// TIA Portal V15.1 export
// export: Created 2024-06-21T08:41:01.6474151Z, ExportSetting WithDefaults, DisplayName Totally Integrated Automation Portal, DisplayVersion V15.1 Update 5, DisplayName TIA Portal Openness, DisplayVersion V15.1 Update 5, DisplayName SINAMICS Startdrive Advanced, DisplayVersion V15.1, DisplayName G130, G150, S120, S150, SINAMICS MV, S210, DisplayVersion V15.1, DisplayName G110M, G120, G120C, G120D, G120P, DisplayVersion V15.1, DisplayName STEP 7 Professional, DisplayVersion V15.1 Update 5, DisplayName STEP 7 Safety, DisplayVersion V15.1, DisplayName WinCC Professional, DisplayVersion V15.1 Update 5, DisplayName SIMATIC Visualization Architect, DisplayVersion V15.1
FUNCTION_BLOCK "LActiveShift"   // FB1800, FBD
TITLE = LActifShift
{ S7_Optimized_Access := 'FALSE' }
AUTHOR : VCC
FAMILY : Supervis
NAME : LActShif
VERSION : 1.0
// ================================================================================
// Module used to give which shift is active with the calendar variable of PLC
// Morning shift: start - stop is defined by HMI
// Evening shift: start - stop is defined by HMI
// Night shift  : start - stop is defined by HMI
// ================================================================================
// stored: AutoNumber false, IsIECCheckEnabled false, SetENOAutomatically False, UDAEnableTagReadback false
   VAR_OUTPUT
      O_MorningShift { ExternalAccessible := 'False'; ExternalVisible := 'False'; ExternalWritable := 'False'} : Bool;   // Morning shift
      O_EveningShift { ExternalAccessible := 'False'; ExternalVisible := 'False'; ExternalWritable := 'False'} : Bool;   // Evening shift
      O_NightShift { ExternalAccessible := 'False'; ExternalVisible := 'False'; ExternalWritable := 'False'} : Bool;   // NightShift
      O_NewShift { ExternalAccessible := 'False'; ExternalVisible := 'False'; ExternalWritable := 'False'} : Bool;   // NewShift / Morning shift
      O_ShiftOverview { ExternalAccessible := 'False'; ExternalVisible := 'False'; ExternalWritable := 'False'} : Struct   // Overview Active Shift
         MorningShift_Day1 { ExternalAccessible := 'False'; ExternalVisible := 'False'; ExternalWritable := 'False'} : Bool;   // Morning Shift of Day 1 (Monday)
         EveningShift_Day1 { ExternalAccessible := 'False'; ExternalVisible := 'False'; ExternalWritable := 'False'} : Bool;   // Evening Shift of Day 1 (Monday)
         NightShift_Day1 { ExternalAccessible := 'False'; ExternalVisible := 'False'; ExternalWritable := 'False'} : Bool;   // Night Shift of Day 1 (Monday-Tuesday)
         MorningShift_Day2 { ExternalAccessible := 'False'; ExternalVisible := 'False'; ExternalWritable := 'False'} : Bool;   // Morning Shift of Day 2 (Tuesday)
         EveningShift_Day2 { ExternalAccessible := 'False'; ExternalVisible := 'False'; ExternalWritable := 'False'} : Bool;   // Evening Shift of Day 2 (Tuesday)
         NightShift_Day2 { ExternalAccessible := 'False'; ExternalVisible := 'False'; ExternalWritable := 'False'} : Bool;   // Night Shift of Day 2 (Tuesday-Wednesday)
         MorningShift_Day3 { ExternalAccessible := 'False'; ExternalVisible := 'False'; ExternalWritable := 'False'} : Bool;   // Morning Shift of Day 3 (Wednesday)
         EveningShift_Day3 { ExternalAccessible := 'False'; ExternalVisible := 'False'; ExternalWritable := 'False'} : Bool;   // Evening Shift of Day 3 (Wednesday)
         NightShift_Day3 { ExternalAccessible := 'False'; ExternalVisible := 'False'; ExternalWritable := 'False'} : Bool;   // night Shift of Day 3 (Wednesday-Thursday)
         MorningShift_Day4 { ExternalAccessible := 'False'; ExternalVisible := 'False'; ExternalWritable := 'False'} : Bool;   // Morning Shift of Day 4 (Thursday)
         EveningShift_Day4 { ExternalAccessible := 'False'; ExternalVisible := 'False'; ExternalWritable := 'False'} : Bool;   // Evening Shift of Day 4 (Thursday)
         NightShift_Day4 { ExternalAccessible := 'False'; ExternalVisible := 'False'; ExternalWritable := 'False'} : Bool;   // Night Shift of Day 4 (Thursday-Friday)
         MorningShift_Day5 { ExternalAccessible := 'False'; ExternalVisible := 'False'; ExternalWritable := 'False'} : Bool;   // Morning Shift of Day 5 (Friday)
         EveningShift_Day5 { ExternalAccessible := 'False'; ExternalVisible := 'False'; ExternalWritable := 'False'} : Bool;   // Evening Shift of Day 5 (Friday)
         NightShift_Day5 { ExternalAccessible := 'False'; ExternalVisible := 'False'; ExternalWritable := 'False'} : Bool;   // Night Shift of Day 5 (Friday-Saturday)
         MorningShift_Day6 { ExternalAccessible := 'False'; ExternalVisible := 'False'; ExternalWritable := 'False'} : Bool;   // Morning Shift of Day 6 (Saturday)
         EveningShift_Day6 { ExternalAccessible := 'False'; ExternalVisible := 'False'; ExternalWritable := 'False'} : Bool;   // Evening Shift of Day 6 (Saturday)
         NightShift_Day6 { ExternalAccessible := 'False'; ExternalVisible := 'False'; ExternalWritable := 'False'} : Bool;   // Night Shift of Day 6 (Saturday-Sunday)
         MorningShift_Day7 { ExternalAccessible := 'False'; ExternalVisible := 'False'; ExternalWritable := 'False'} : Bool;   // Morning Shift of Day 7 (Sunday)
         EveningShift_Day7 { ExternalAccessible := 'False'; ExternalVisible := 'False'; ExternalWritable := 'False'} : Bool;   // Evening Shift of Day 7 (Sunday)
         NightShift_Day7 { ExternalAccessible := 'False'; ExternalVisible := 'False'; ExternalWritable := 'False'} : Bool;   // night Shift of Day 7 (Sunday-Monday)
      END_STRUCT;
      H_IAnim { ExternalAccessible := 'False'; ExternalVisible := 'False'; ExternalWritable := 'False'} : Word;   // HMI Animation of the icon
   END_VAR
   VAR DB_SPECIFIC
      H_In : Struct   // HMI
         StartMorningDay1 : Real := 5.15;   // Start time of morning shift - Day 1
         StartEveningDay1 : Real := 13.15;   // Start time of evening shift - Day 1
         StartNightDay1 : Real := 21.15;   // Start time of night shift - Day 1
         StartMorningDay2 : Real := 5.15;   // Start time of morning shift - Day 2
         StartEveningDay2 : Real := 13.15;   // Start time of evening shift - Day 2
         StartNightDay2 : Real := 21.15;   // Start time of night shift - Day 2
         StartMorningDay3 : Real := 5.15;   // Start time of morning shift - Day 3
         StartEveningDay3 : Real := 13.15;   // Start time of evening shift - Day 3
         StartNightDay3 : Real := 21.15;   // Start time of night shift - Day 3
         StartMorningDay4 : Real := 5.15;   // Start time of morning shift - Day 4
         StartEveningDay4 : Real := 13.15;   // Start time of evening shift - Day 4
         StartNightDay4 : Real := 21.15;   // Start time of night shift - Day 4
         StartMorningDay5 : Real := 5.15;   // Start time of morning shift - Day 5
         StartEveningDay5 : Real := 12.25;   // Start time of evening shift - Day 5
         StartNightDay5 : Real := 19.35;   // Start time of night shift - Day 5
         StartMorningDay6 : Real := 5.15;   // Start time of morning shift - Day 6
         StartEveningDay6 : Real := 13.15;   // Start time of evening shift - Day 6
         StartNightDay6 : Real := 21.15;   // Start time of night shift - Day 6
         StartMorningDay7 : Real := 5.15;   // Start time of morning shift - Day 7
         StartEveningDay7 : Real := 13.15;   // Start time of evening shift - Day 7
         StartNightDay7 : Real := 21.15;   // Start time of night shift - Day 7
      END_STRUCT;
      H_Out : Struct   // HMI
         Anim : Word;   // HMI Animation of the object
         DBnr : Int;   // HMI Animation DB number
      END_STRUCT;
      MorningShift_Day1 { ExternalAccessible := 'False'; ExternalVisible := 'False'; ExternalWritable := 'False'} : Bool;   // Morning Shift of Day 1 (Monday)
      EveningShift_Day1 { ExternalAccessible := 'False'; ExternalVisible := 'False'; ExternalWritable := 'False'} : Bool;   // Evening Shift of Day 1 (Monday)
      NightShift_Day1 { ExternalAccessible := 'False'; ExternalVisible := 'False'; ExternalWritable := 'False'} : Bool;   // Night Shift of Day 1 (Monday-Tuesday)
      MorningShift_Day2 { ExternalAccessible := 'False'; ExternalVisible := 'False'; ExternalWritable := 'False'} : Bool;   // Morning Shift of Day 2 (Tuesday)
      EveningShift_Day2 { ExternalAccessible := 'False'; ExternalVisible := 'False'; ExternalWritable := 'False'} : Bool;   // Evening Shift of Day 2 (Tuesday)
      NightShift_Day2 { ExternalAccessible := 'False'; ExternalVisible := 'False'; ExternalWritable := 'False'} : Bool;   // Night Shift of Day 2 (Tuesday-Wednesday)
      MorningShift_Day3 { ExternalAccessible := 'False'; ExternalVisible := 'False'; ExternalWritable := 'False'} : Bool;   // Morning Shift of Day 3 (Wednesday)
      EveningShift_Day3 { ExternalAccessible := 'False'; ExternalVisible := 'False'; ExternalWritable := 'False'} : Bool;   // Evening Shift of Day 3 (Wednesday)
      NightShift_Day3 { ExternalAccessible := 'False'; ExternalVisible := 'False'; ExternalWritable := 'False'} : Bool;   // night Shift of Day 3 (Wednesday-Thursday)
      MorningShift_Day4 { ExternalAccessible := 'False'; ExternalVisible := 'False'; ExternalWritable := 'False'} : Bool;   // Morning Shift of Day 4 (Thursday)
      EveningShift_Day4 { ExternalAccessible := 'False'; ExternalVisible := 'False'; ExternalWritable := 'False'} : Bool;   // Evening Shift of Day 4 (Thursday)
      NightShift_Day4 { ExternalAccessible := 'False'; ExternalVisible := 'False'; ExternalWritable := 'False'} : Bool;   // Night Shift of Day 4 (Thursday-Friday)
      MorningShift_Day5 { ExternalAccessible := 'False'; ExternalVisible := 'False'; ExternalWritable := 'False'} : Bool;   // Morning Shift of Day 5 (Friday)
      EveningShift_Day5 { ExternalAccessible := 'False'; ExternalVisible := 'False'; ExternalWritable := 'False'} : Bool;   // Evening Shift of Day 5 (Friday)
      NightShift_Day5 { ExternalAccessible := 'False'; ExternalVisible := 'False'; ExternalWritable := 'False'} : Bool;   // Night Shift of Day 5 (Friday-Saturday)
      MorningShift_Day6 { ExternalAccessible := 'False'; ExternalVisible := 'False'; ExternalWritable := 'False'} : Bool;   // Morning Shift of Day 6 (Saturday)
      EveningShift_Day6 { ExternalAccessible := 'False'; ExternalVisible := 'False'; ExternalWritable := 'False'} : Bool;   // Evening Shift of Day 6 (Saturday)
      NightShift_Day6 { ExternalAccessible := 'False'; ExternalVisible := 'False'; ExternalWritable := 'False'} : Bool;   // Night Shift of Day 6 (Saturday-Sunday)
      MorningShift_Day7 { ExternalAccessible := 'False'; ExternalVisible := 'False'; ExternalWritable := 'False'} : Bool;   // Morning Shift of Day 7 (Sunday)
      EveningShift_Day7 { ExternalAccessible := 'False'; ExternalVisible := 'False'; ExternalWritable := 'False'} : Bool;   // Evening Shift of Day 7 (Sunday)
      NightShift_Day7 { ExternalAccessible := 'False'; ExternalVisible := 'False'; ExternalWritable := 'False'} : Bool;   // night Shift of Day 7 (Sunday-Monday)
      MorningShift { ExternalAccessible := 'False'; ExternalVisible := 'False'; ExternalWritable := 'False'} : Bool;   // Morning shift
      EveningShift { ExternalAccessible := 'False'; ExternalVisible := 'False'; ExternalWritable := 'False'} : Bool;   // Evening shift
      NightShift { ExternalAccessible := 'False'; ExternalVisible := 'False'; ExternalWritable := 'False'} : Bool;   // NightShift
      NewShift { ExternalAccessible := 'False'; ExternalVisible := 'False'; ExternalWritable := 'False'} : Bool;   // NewShift / Morning shift
      NewMorningShiftTrig { ExternalAccessible := 'False'; ExternalVisible := 'False'; ExternalWritable := 'False'} : Bool;   // Trigger for New Morning shift / Morning shift
      NewEveningShiftTrig { ExternalAccessible := 'False'; ExternalVisible := 'False'; ExternalWritable := 'False'} : Bool;   // Trigger for New Evening shift / Evening shift
      NewNightShiftTrig { ExternalAccessible := 'False'; ExternalVisible := 'False'; ExternalWritable := 'False'} : Bool;   // Trigger for New NightShift / NightShift
      Day1 { ExternalAccessible := 'False'; ExternalVisible := 'False'; ExternalWritable := 'False'} : Bool;   // Day 1 = Monday
      Day2 { ExternalAccessible := 'False'; ExternalVisible := 'False'; ExternalWritable := 'False'} : Bool;   // Day 2 = Tuesday
      Day3 { ExternalAccessible := 'False'; ExternalVisible := 'False'; ExternalWritable := 'False'} : Bool;   // Day 3 = Wednesday
      Day4 { ExternalAccessible := 'False'; ExternalVisible := 'False'; ExternalWritable := 'False'} : Bool;   // Day 4 = Thursday
      Day5 { ExternalAccessible := 'False'; ExternalVisible := 'False'; ExternalWritable := 'False'} : Bool;   // Day 5 = Friday
      Day6 { ExternalAccessible := 'False'; ExternalVisible := 'False'; ExternalWritable := 'False'} : Bool;   // Day 6 = Saturday
      Day7 { ExternalAccessible := 'False'; ExternalVisible := 'False'; ExternalWritable := 'False'} : Bool;   // Day 7 = Sunday
      Day1_Int_Morning { ExternalAccessible := 'False'; ExternalVisible := 'False'; ExternalWritable := 'False'} : Int := 515;   // Start integer of morning shift - Day 1
      Day1_Int_Evening { ExternalAccessible := 'False'; ExternalVisible := 'False'; ExternalWritable := 'False'} : Int := 1315;   // Start integer of evening shift - Day 1
      Day1_Int_Night { ExternalAccessible := 'False'; ExternalVisible := 'False'; ExternalWritable := 'False'} : Int := 2115;   // Start integer of night shift - Day 1
      Day2_Int_Morning { ExternalAccessible := 'False'; ExternalVisible := 'False'; ExternalWritable := 'False'} : Int := 515;   // Start integer of morning shift - Day 2
      Day2_Int_Evening { ExternalAccessible := 'False'; ExternalVisible := 'False'; ExternalWritable := 'False'} : Int := 1315;   // Start integer of evening shift - Day 2
      Day2_Int_Night { ExternalAccessible := 'False'; ExternalVisible := 'False'; ExternalWritable := 'False'} : Int := 2115;   // Start integer of night shift - Day 2
      Day3_Int_Morning { ExternalAccessible := 'False'; ExternalVisible := 'False'; ExternalWritable := 'False'} : Int := 515;   // Start integer of morning shift - Day 3
      Day3_Int_Evening { ExternalAccessible := 'False'; ExternalVisible := 'False'; ExternalWritable := 'False'} : Int := 1315;   // Start integer of evening shift - Day 3
      Day3_Int_Night { ExternalAccessible := 'False'; ExternalVisible := 'False'; ExternalWritable := 'False'} : Int := 2115;   // Start integer of night shift - Day 3
      Day4_Int_Morning { ExternalAccessible := 'False'; ExternalVisible := 'False'; ExternalWritable := 'False'} : Int := 515;   // Start integer of morning shift - Day 4
      Day4_Int_Evening { ExternalAccessible := 'False'; ExternalVisible := 'False'; ExternalWritable := 'False'} : Int := 1315;   // Start integer of evening shift - Day 4
      Day4_Int_Night { ExternalAccessible := 'False'; ExternalVisible := 'False'; ExternalWritable := 'False'} : Int := 2115;   // Start integer of night shift - Day 4
      Day5_Int_Morning { ExternalAccessible := 'False'; ExternalVisible := 'False'; ExternalWritable := 'False'} : Int := 515;   // Start integer of morning shift - Day 5
      Day5_Int_Evening { ExternalAccessible := 'False'; ExternalVisible := 'False'; ExternalWritable := 'False'} : Int := 1225;   // Start integer of evening shift - Day 5
      Day5_Int_Night { ExternalAccessible := 'False'; ExternalVisible := 'False'; ExternalWritable := 'False'} : Int := 1935;   // Start integer of night shift - Day 5
      Day6_Int_Morning { ExternalAccessible := 'False'; ExternalVisible := 'False'; ExternalWritable := 'False'} : Int := 515;   // Start integer of morning shift - Day 6
      Day6_Int_Evening { ExternalAccessible := 'False'; ExternalVisible := 'False'; ExternalWritable := 'False'} : Int := 1315;   // Start integer of evening shift - Day 6
      Day6_Int_Night { ExternalAccessible := 'False'; ExternalVisible := 'False'; ExternalWritable := 'False'} : Int := 2115;   // Start integer of night shift - Day 6
      Day7_Int_Morning { ExternalAccessible := 'False'; ExternalVisible := 'False'; ExternalWritable := 'False'} : Int := 515;   // Start integer of morning shift - Day 7
      Day7_Int_Evening { ExternalAccessible := 'False'; ExternalVisible := 'False'; ExternalWritable := 'False'} : Int := 1315;   // Start integer of evening shift - Day 7
      Day7_Int_Night { ExternalAccessible := 'False'; ExternalVisible := 'False'; ExternalWritable := 'False'} : Int := 2115;   // Start integer of night shift - Day 7
      DBnr { ExternalAccessible := 'False'; ExternalVisible := 'False'; ExternalWritable := 'False'} : Int;   // HMI DB number
   END_VAR
   VAR_TEMP
      Temp1 : Real;
      Temp2 : Int;
   END_VAR
   VAR_TEMP   // added for the SCL form of the ladder/FBD networks
      _w1 : Bool;
      _w2 : Bool;
      _w3 : Bool;
   END_VAR
BEGIN

NETWORK
TITLE = **** 1 - Inputs **** DB number
// DB number
      L     DINO;
      T     #DBnr;

NETWORK
TITLE = **** 4.4 - Machine status - Calculated **** Copy time from HMI to integer
// Copy time from HMI to integer
//********************** Time day 1 *****************************
      L     #H_In.StartMorningDay1;  // Load Start time of morning shift - Day 1
      L     100.0;  // * 100
      *R;  // *
      RND;  // Conversion real to integer
      T     #Day1_Int_Morning;  // Load start time of morning shift = Day 1

      L     #H_In.StartEveningDay1;  // Load Start time of evening shift - Day 1
      L     100.0;  // * 100
      *R;  // *
      RND;  // Conversion real to integer
      T     #Day1_Int_Evening;  // Load start time of evening shift = Day 1

      L     #H_In.StartNightDay1;  // Load Start time of night shift - Day 1
      L     100.0;  // * 100
      *R;  // *
      RND;  // Conversion real to integer
      T     #Day1_Int_Night;  // Load start time of night shift = Day 1


//********************** Time day 2 *****************************
      L     #H_In.StartMorningDay2;  // Load Start time of morning shift - Day 2
      L     100.0;  // * 100
      *R;  // *
      RND;  // Conversion real to integer
      T     #Day2_Int_Morning;  // Load start time of morning shift = Day 2

      L     #H_In.StartEveningDay2;  // Load Start time of evening shift - Day 2
      L     100.0;  // * 100
      *R;  // *
      RND;  // Conversion real to integer
      T     #Day2_Int_Evening;  // Load start time of evening shift = Day 2

      L     #H_In.StartNightDay2;  // Load Start time of night shift - Day 2
      L     100.0;  // * 100
      *R;  // *
      RND;  // Conversion real to integer
      T     #Day2_Int_Night;  // Load start time of night shift = Day 2

//********************** Time day 3 *****************************
      L     #H_In.StartMorningDay3;  // Load Start time of morning shift - Day 3
      L     100.0;  // * 100
      *R;  // *
      RND;  // Conversion real to integer
      T     #Day3_Int_Morning;  // Load start time of morning shift = Day 3

      L     #H_In.StartEveningDay3;  // Load Start time of evening shift - Day 3
      L     100.0;  // * 100
      *R;  // *
      RND;  // Conversion real to integer
      T     #Day3_Int_Evening;  // Load start time of evening shift = Day 3

      L     #H_In.StartNightDay3;  // Load Start time of night shift - Day 3
      L     100.0;  // * 100
      *R;  // *
      RND;  // Conversion real to integer
      T     #Day3_Int_Night;  // Load start time of night shift = Day 3

//********************** Time day 4 *****************************
      L     #H_In.StartMorningDay4;  // Load Start time of morning shift - Day 4
      L     100.0;  // * 100
      *R;  // *
      RND;  // Conversion real to integer
      T     #Day4_Int_Morning;  // Load start time of morning shift = Day 4

      L     #H_In.StartEveningDay4;  // Load Start time of evening shift - Day 4
      L     100.0;  // * 100
      *R;  // *
      RND;  // Conversion real to integer
      T     #Day4_Int_Evening;  // Load start time of evening shift = Day 4

      L     #H_In.StartNightDay4;  // Load Start time of night shift - Day 4
      L     100.0;  // * 100
      *R;  // *
      RND;  // Conversion real to integer
      T     #Day4_Int_Night;  // Load start time of night shift = Day 4

//********************** Time day 5 *****************************
      L     #H_In.StartMorningDay5;  // Load Start time of morning shift - Day 5
      L     100.0;  // * 100
      *R;  // *
      RND;  // Conversion real to integer
      T     #Day5_Int_Morning;  // Load start time of morning shift = Day 5

      L     #H_In.StartEveningDay5;  // Load Start time of evening shift - Day 5
      L     100.0;  // * 100
      *R;  // *
      RND;  // Conversion real to integer
      T     #Day5_Int_Evening;  // Load start time of evening shift = Day 5

      L     #H_In.StartNightDay5;  // Load Start time of night shift - Day 5
      L     100.0;  // * 100
      *R;  // *
      RND;  // Conversion real to integer
      T     #Day5_Int_Night;  // Load start time of night shift = Day 5

//********************** Time day 6 *****************************
      L     #H_In.StartMorningDay6;  // Load Start time of morning shift - Day 6
      L     100.0;  // * 100
      *R;  // *
      RND;  // Conversion real to integer
      T     #Day6_Int_Morning;  // Load start time of morning shift = Day 6

      L     #H_In.StartEveningDay6;  // Load Start time of evening shift - Day 6
      L     100.0;  // * 100
      *R;  // *
      RND;  // Conversion real to integer
      T     #Day6_Int_Evening;  // Load start time of evening shift = Day 6

      L     #H_In.StartNightDay6;  // Load Start time of night shift - Day 6
      L     100.0;  // * 100
      *R;  // *
      RND;  // Conversion real to integer
      T     #Day6_Int_Night;  // Load start time of night shift = Day 6

//********************** Time day 7 *****************************
      L     #H_In.StartMorningDay7;  // Load Start time of morning shift - Day 7
      L     100.0;  // * 100
      *R;  // *
      RND;  // Conversion real to integer
      T     #Day7_Int_Morning;  // Load start time of morning shift = Day 7

      L     #H_In.StartEveningDay7;  // Load Start time of evening shift - Day 7
      L     100.0;  // * 100
      *R;  // *
      RND;  // Conversion real to integer
      T     #Day7_Int_Evening;  // Load start time of evening shift = Day 7

      L     #H_In.StartNightDay7;  // Load Start time of night shift - Day 7
      L     100.0;  // * 100
      *R;  // *
      RND;  // Conversion real to integer
      T     #Day7_Int_Night;  // Load start time of night shift = Day 7

REGION Network 3: **** 4.4 - Machine status - Calculated **** Morning Shift of Day 1
   // Morning Shift of Day 1
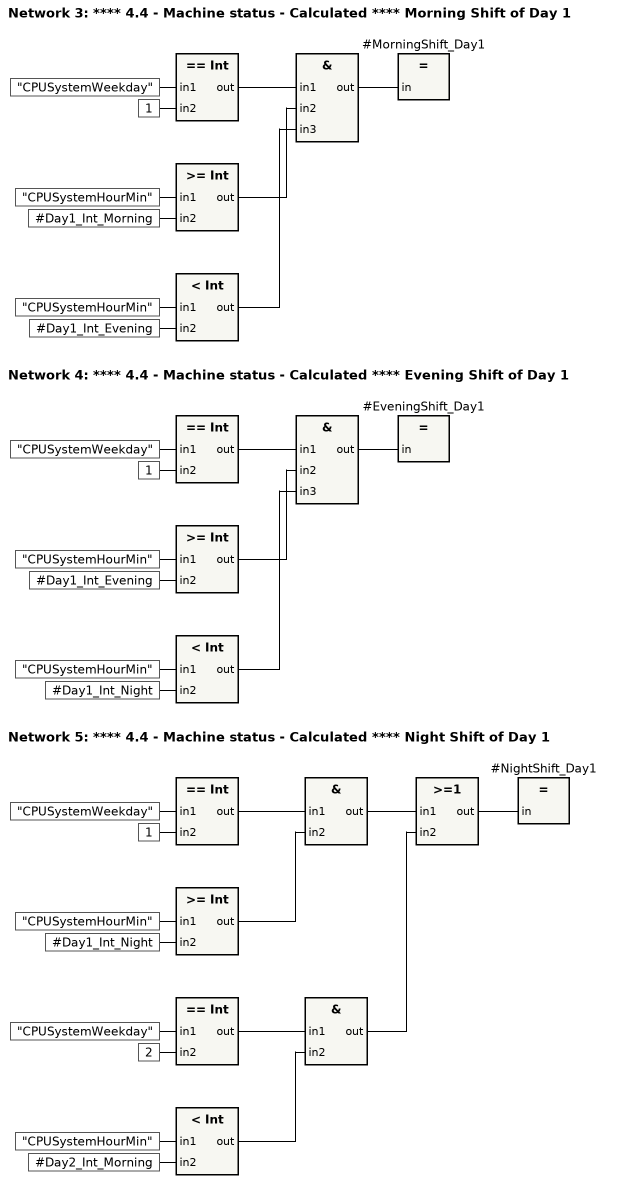
   #MorningShift_Day1 := ("CPUSystemWeekday" = 1) AND ("CPUSystemHourMin" >= #Day1_Int_Morning) AND ("CPUSystemHourMin" < #Day1_Int_Evening);
END_REGION

REGION Network 4: **** 4.4 - Machine status - Calculated **** Evening Shift of Day 1
   // Evening Shift of Day 1
   #EveningShift_Day1 := ("CPUSystemWeekday" = 1) AND ("CPUSystemHourMin" >= #Day1_Int_Evening) AND ("CPUSystemHourMin" < #Day1_Int_Night);
END_REGION

REGION Network 5: **** 4.4 - Machine status - Calculated **** Night Shift of Day 1
   // Night Shift of Day 1
   #NightShift_Day1 := (("CPUSystemWeekday" = 1) AND ("CPUSystemHourMin" >= #Day1_Int_Night)) OR (("CPUSystemWeekday" = 2) AND ("CPUSystemHourMin" < #Day2_Int_Morning));
END_REGION

REGION Network 6: **** 4.4 - Machine status - Calculated **** Morning Shift of Day 2
   // Morning Shift of Day 2
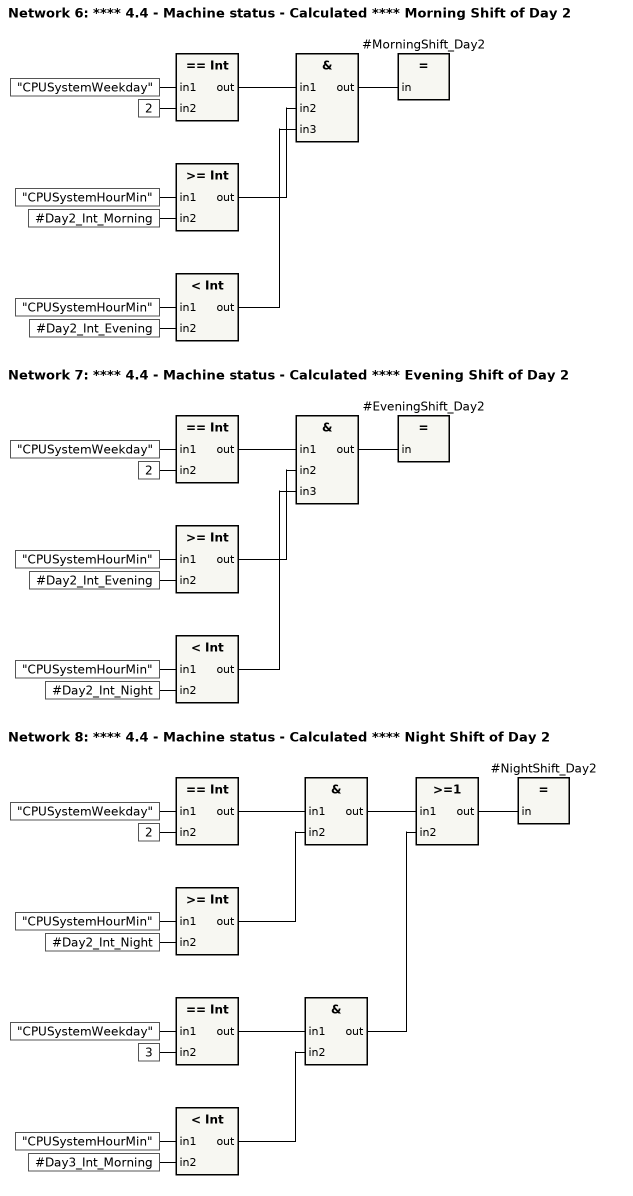
   #MorningShift_Day2 := ("CPUSystemWeekday" = 2) AND ("CPUSystemHourMin" >= #Day2_Int_Morning) AND ("CPUSystemHourMin" < #Day2_Int_Evening);
END_REGION

REGION Network 7: **** 4.4 - Machine status - Calculated **** Evening Shift of Day 2
   // Evening Shift of Day 2
   #EveningShift_Day2 := ("CPUSystemWeekday" = 2) AND ("CPUSystemHourMin" >= #Day2_Int_Evening) AND ("CPUSystemHourMin" < #Day2_Int_Night);
END_REGION

REGION Network 8: **** 4.4 - Machine status - Calculated **** Night Shift of Day 2
   // Night Shift of Day 2
   #NightShift_Day2 := (("CPUSystemWeekday" = 2) AND ("CPUSystemHourMin" >= #Day2_Int_Night)) OR (("CPUSystemWeekday" = 3) AND ("CPUSystemHourMin" < #Day3_Int_Morning));
END_REGION

REGION Network 9: **** 4.4 - Machine status - Calculated **** Morning Shift of Day 3
   // Morning Shift of Day 3
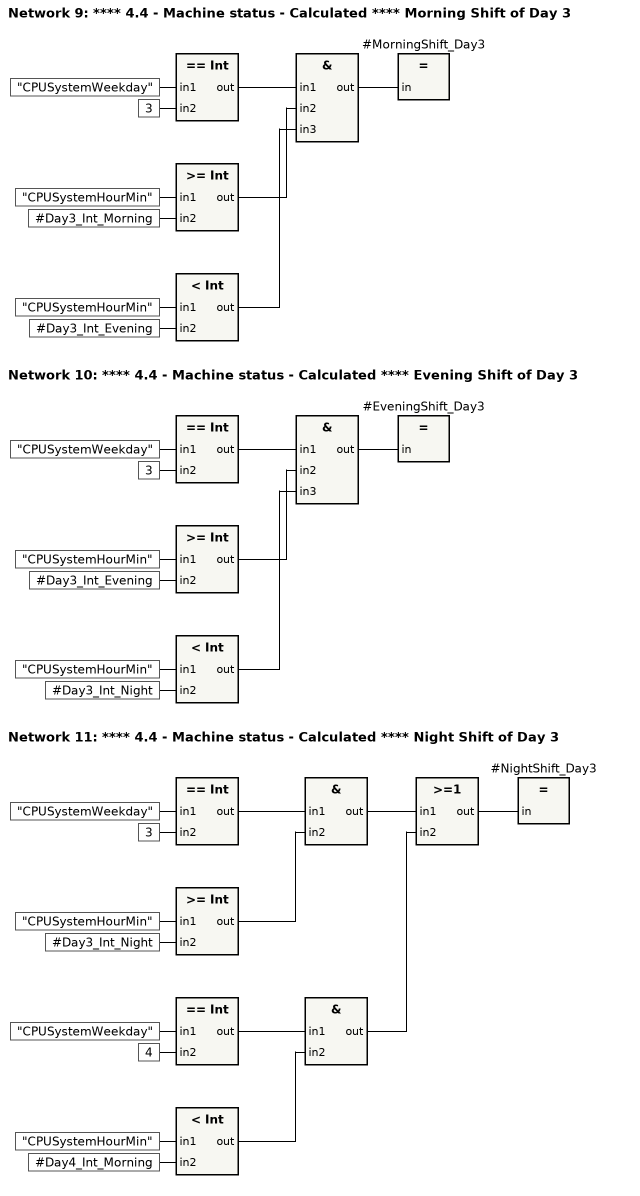
   #MorningShift_Day3 := ("CPUSystemWeekday" = 3) AND ("CPUSystemHourMin" >= #Day3_Int_Morning) AND ("CPUSystemHourMin" < #Day3_Int_Evening);
END_REGION

REGION Network 10: **** 4.4 - Machine status - Calculated **** Evening Shift of Day 3
   // Evening Shift of Day 3
   #EveningShift_Day3 := ("CPUSystemWeekday" = 3) AND ("CPUSystemHourMin" >= #Day3_Int_Evening) AND ("CPUSystemHourMin" < #Day3_Int_Night);
END_REGION

REGION Network 11: **** 4.4 - Machine status - Calculated **** Night Shift of Day 3
   // Night Shift of Day 3
   #NightShift_Day3 := (("CPUSystemWeekday" = 3) AND ("CPUSystemHourMin" >= #Day3_Int_Night)) OR (("CPUSystemWeekday" = 4) AND ("CPUSystemHourMin" < #Day4_Int_Morning));
END_REGION

REGION Network 12: **** 4.4 - Machine status - Calculated **** Morning Shift of Day 4
   // Morning Shift of Day 4
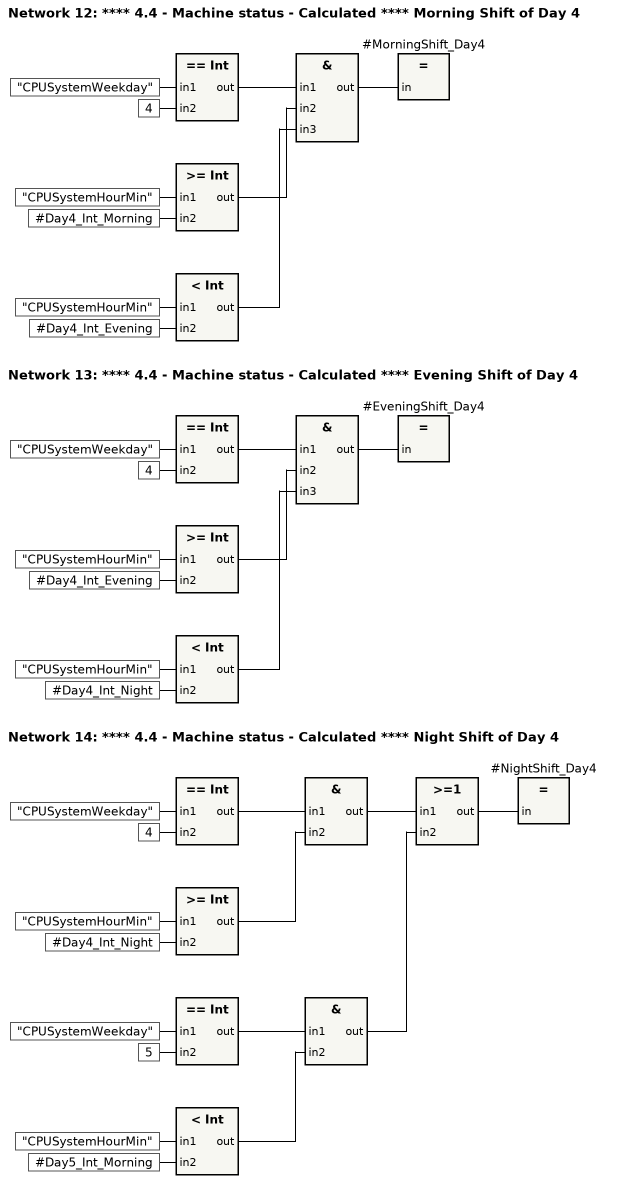
   #MorningShift_Day4 := ("CPUSystemWeekday" = 4) AND ("CPUSystemHourMin" >= #Day4_Int_Morning) AND ("CPUSystemHourMin" < #Day4_Int_Evening);
END_REGION

REGION Network 13: **** 4.4 - Machine status - Calculated **** Evening Shift of Day 4
   // Evening Shift of Day 4
   #EveningShift_Day4 := ("CPUSystemWeekday" = 4) AND ("CPUSystemHourMin" >= #Day4_Int_Evening) AND ("CPUSystemHourMin" < #Day4_Int_Night);
END_REGION

REGION Network 14: **** 4.4 - Machine status - Calculated **** Night Shift of Day 4
   // Night Shift of Day 4
   #NightShift_Day4 := (("CPUSystemWeekday" = 4) AND ("CPUSystemHourMin" >= #Day4_Int_Night)) OR (("CPUSystemWeekday" = 5) AND ("CPUSystemHourMin" < #Day5_Int_Morning));
END_REGION

REGION Network 15: **** 4.4 - Machine status - Calculated **** Morning Shift of Day 5
   // Morning Shift of Day 5
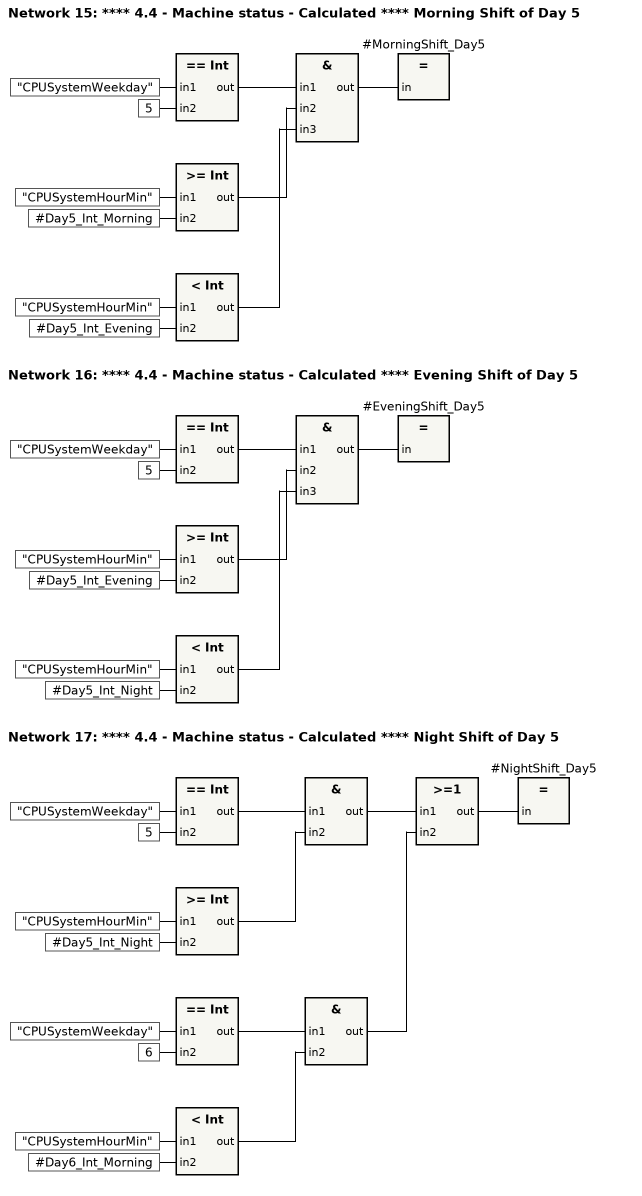
   #MorningShift_Day5 := ("CPUSystemWeekday" = 5) AND ("CPUSystemHourMin" >= #Day5_Int_Morning) AND ("CPUSystemHourMin" < #Day5_Int_Evening);
END_REGION

REGION Network 16: **** 4.4 - Machine status - Calculated **** Evening Shift of Day 5
   // Evening Shift of Day 5
   #EveningShift_Day5 := ("CPUSystemWeekday" = 5) AND ("CPUSystemHourMin" >= #Day5_Int_Evening) AND ("CPUSystemHourMin" < #Day5_Int_Night);
END_REGION

REGION Network 17: **** 4.4 - Machine status - Calculated **** Night Shift of Day 5
   // Night Shift of Day 5
   #NightShift_Day5 := (("CPUSystemWeekday" = 5) AND ("CPUSystemHourMin" >= #Day5_Int_Night)) OR (("CPUSystemWeekday" = 6) AND ("CPUSystemHourMin" < #Day6_Int_Morning));
END_REGION

REGION Network 18: **** 4.4 - Machine status - Calculated **** Morning Shift of Day 6
   // Morning Shift of Day 6
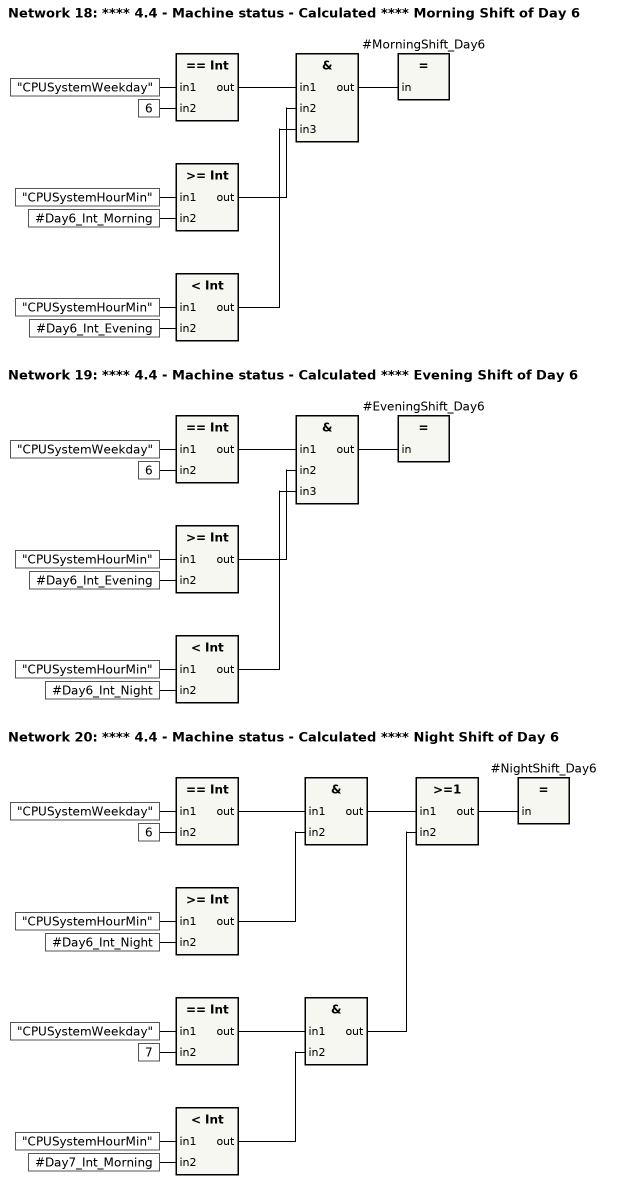
   #MorningShift_Day6 := ("CPUSystemWeekday" = 6) AND ("CPUSystemHourMin" >= #Day6_Int_Morning) AND ("CPUSystemHourMin" < #Day6_Int_Evening);
END_REGION

REGION Network 19: **** 4.4 - Machine status - Calculated **** Evening Shift of Day 6
   // Evening Shift of Day 6
   #EveningShift_Day6 := ("CPUSystemWeekday" = 6) AND ("CPUSystemHourMin" >= #Day6_Int_Evening) AND ("CPUSystemHourMin" < #Day6_Int_Night);
END_REGION

REGION Network 20: **** 4.4 - Machine status - Calculated **** Night Shift of Day 6
   // Night Shift of Day 6
   #NightShift_Day6 := (("CPUSystemWeekday" = 6) AND ("CPUSystemHourMin" >= #Day6_Int_Night)) OR (("CPUSystemWeekday" = 7) AND ("CPUSystemHourMin" < #Day7_Int_Morning));
END_REGION

REGION Network 21: **** 4.4 - Machine status - Calculated **** Morning Shift of Day 7
   // Morning Shift of Day 7
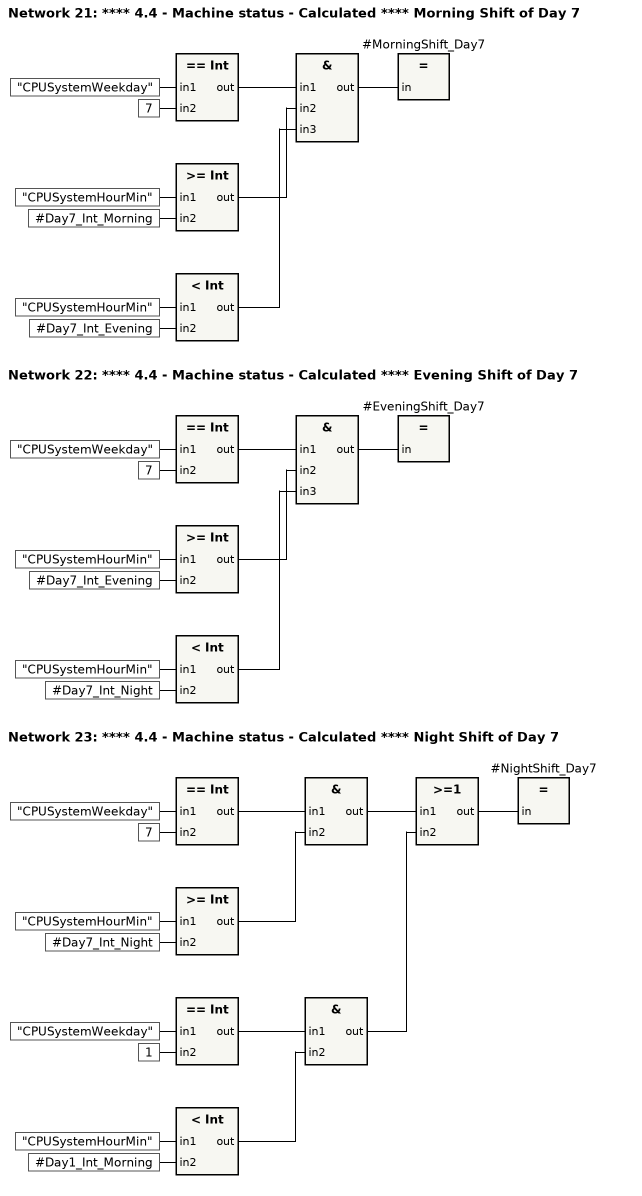
   #MorningShift_Day7 := ("CPUSystemWeekday" = 7) AND ("CPUSystemHourMin" >= #Day7_Int_Morning) AND ("CPUSystemHourMin" < #Day7_Int_Evening);
END_REGION

REGION Network 22: **** 4.4 - Machine status - Calculated **** Evening Shift of Day 7
   // Evening Shift of Day 7
   #EveningShift_Day7 := ("CPUSystemWeekday" = 7) AND ("CPUSystemHourMin" >= #Day7_Int_Evening) AND ("CPUSystemHourMin" < #Day7_Int_Night);
END_REGION

REGION Network 23: **** 4.4 - Machine status - Calculated **** Night Shift of Day 7
   // Night Shift of Day 7
   #NightShift_Day7 := (("CPUSystemWeekday" = 7) AND ("CPUSystemHourMin" >= #Day7_Int_Night)) OR (("CPUSystemWeekday" = 1) AND ("CPUSystemHourMin" < #Day1_Int_Morning));
END_REGION

REGION Network 24: **** 4.4 - Machine status - Calculated **** Morning shift
   // Morning shift
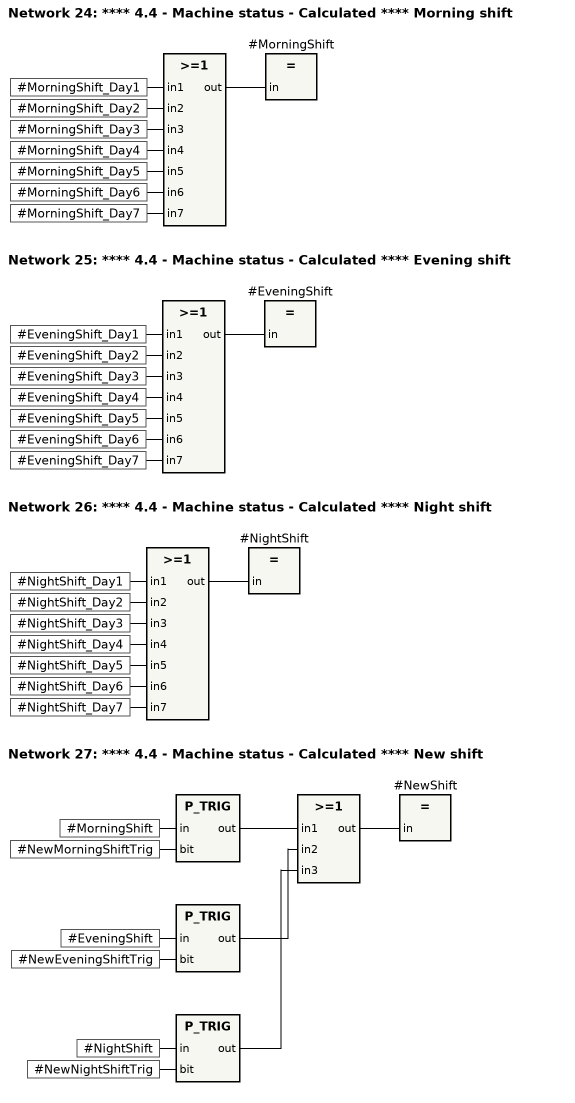
   #MorningShift := #MorningShift_Day1 OR #MorningShift_Day2 OR #MorningShift_Day3 OR #MorningShift_Day4 OR #MorningShift_Day5 OR #MorningShift_Day6 OR #MorningShift_Day7;
END_REGION

REGION Network 25: **** 4.4 - Machine status - Calculated **** Evening shift
   // Evening shift
   #EveningShift := #EveningShift_Day1 OR #EveningShift_Day2 OR #EveningShift_Day3 OR #EveningShift_Day4 OR #EveningShift_Day5 OR #EveningShift_Day6 OR #EveningShift_Day7;
END_REGION

REGION Network 26: **** 4.4 - Machine status - Calculated **** Night shift
   // Night shift
   #NightShift := #NightShift_Day1 OR #NightShift_Day2 OR #NightShift_Day3 OR #NightShift_Day4 OR #NightShift_Day5 OR #NightShift_Day6 OR #NightShift_Day7;
END_REGION

REGION Network 27: **** 4.4 - Machine status - Calculated **** New shift
   #_w1 := #MorningShift AND NOT #NewMorningShiftTrig;   // rising edge
   #NewMorningShiftTrig := #MorningShift;
   #_w2 := #EveningShift AND NOT #NewEveningShiftTrig;   // rising edge
   #NewEveningShiftTrig := #EveningShift;
   #_w3 := #NightShift AND NOT #NewNightShiftTrig;   // rising edge
   #NewNightShiftTrig := #NightShift;
   #NewShift := #_w1 OR #_w2 OR #_w3;
END_REGION

NETWORK
TITLE = **** 4.4 - Machine status - Calculated **** Days of the week
// Days of the week

//Day1
      L     "CPUSystemWeekday";
      L     1;
      ==I;
      =     #Day1;

//Day2
      L     "CPUSystemWeekday";
      L     2;
      ==I;
      =     #Day2;

//Day3
      L     "CPUSystemWeekday";
      L     3;
      ==I;
      =     #Day3;

//Day4
      L     "CPUSystemWeekday";
      L     4;
      ==I;
      =     #Day4;

//Day5
      L     "CPUSystemWeekday";
      L     5;
      ==I;
      =     #Day5;

//Day6
      L     "CPUSystemWeekday";
      L     6;
      ==I;
      =     #Day6;

//Day7
      L     "CPUSystemWeekday";
      L     7;
      ==I;
      =     #Day7;


REGION Network 29: **** 4.6 - Machine status - Indications **** Icon Animation
   // Icon Animation for HMI
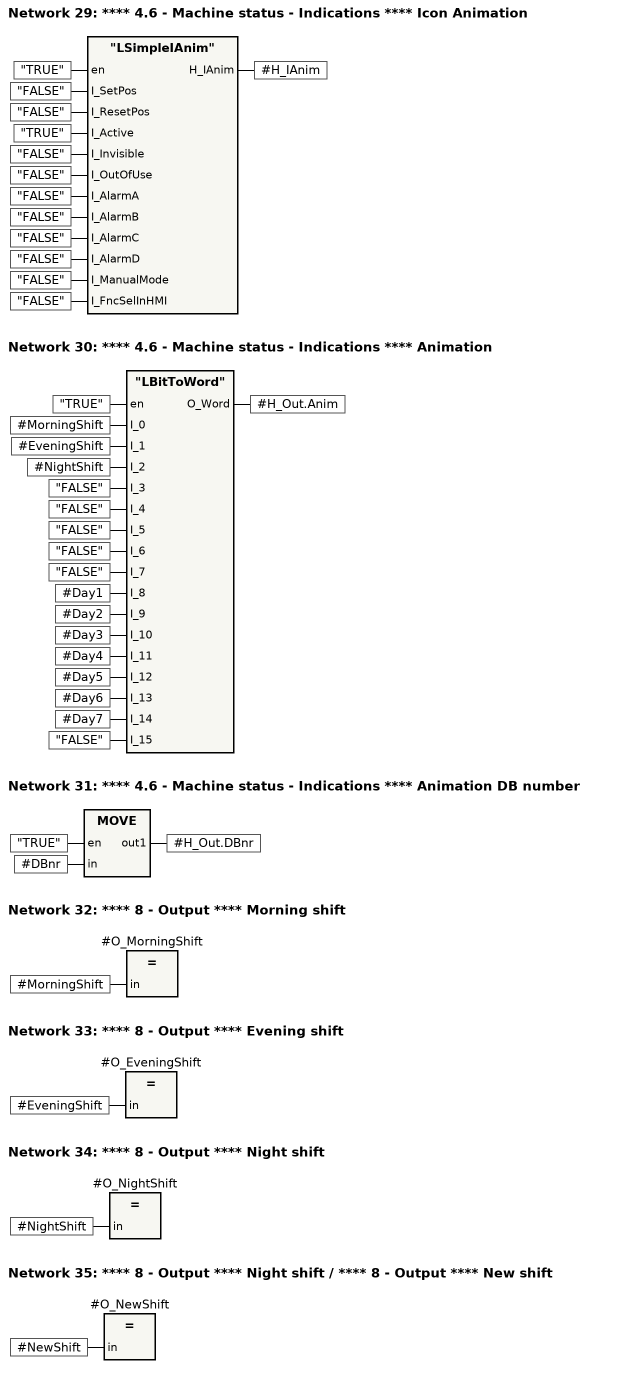
   IF "TRUE" THEN
       "LSimpleIAnim"(I_SetPos := "FALSE",
                      I_ResetPos := "FALSE",
                      I_Active := "TRUE",
                      I_Invisible := "FALSE",
                      I_OutOfUse := "FALSE",
                      I_AlarmA := "FALSE",
                      I_AlarmB := "FALSE",
                      I_AlarmC := "FALSE",
                      I_AlarmD := "FALSE",
                      I_ManualMode := "FALSE",
                      I_FncSelInHMI := "FALSE",
                      H_IAnim => #H_IAnim);
   END_IF;
END_REGION

REGION Network 30: **** 4.6 - Machine status - Indications **** Animation
   // Animation for HMI
   IF "TRUE" THEN
       "LBitToWord"(I_0 := #MorningShift,
                    I_1 := #EveningShift,
                    I_2 := #NightShift,
                    I_3 := "FALSE",
                    I_4 := "FALSE",
                    I_5 := "FALSE",
                    I_6 := "FALSE",
                    I_7 := "FALSE",
                    I_8 := #Day1,
                    I_9 := #Day2,
                    I_10 := #Day3,
                    I_11 := #Day4,
                    I_12 := #Day5,
                    I_13 := #Day6,
                    I_14 := #Day7,
                    I_15 := "FALSE",
                    O_Word => #H_Out.Anim);
   END_IF;
END_REGION

REGION Network 31: **** 4.6 - Machine status - Indications **** Animation DB number
   // Animation DB number
   IF "TRUE" THEN #H_Out.DBnr := #DBnr; END_IF;
END_REGION

REGION Network 32: **** 8 - Output **** Morning shift
   // Morning shift
   #O_MorningShift := #MorningShift;
END_REGION

REGION Network 33: **** 8 - Output **** Evening shift
   // Evening shift
   #O_EveningShift := #EveningShift;
END_REGION

REGION Network 34: **** 8 - Output **** Night shift
   // Night shift
   #O_NightShift := #NightShift;
END_REGION

REGION Network 35: **** 8 - Output **** Night shift / **** 8 - Output **** New shift
   // Night shift
   #O_NewShift := #NewShift;
END_REGION

REGION Network 36: **** 8 - Output **** Active Shift
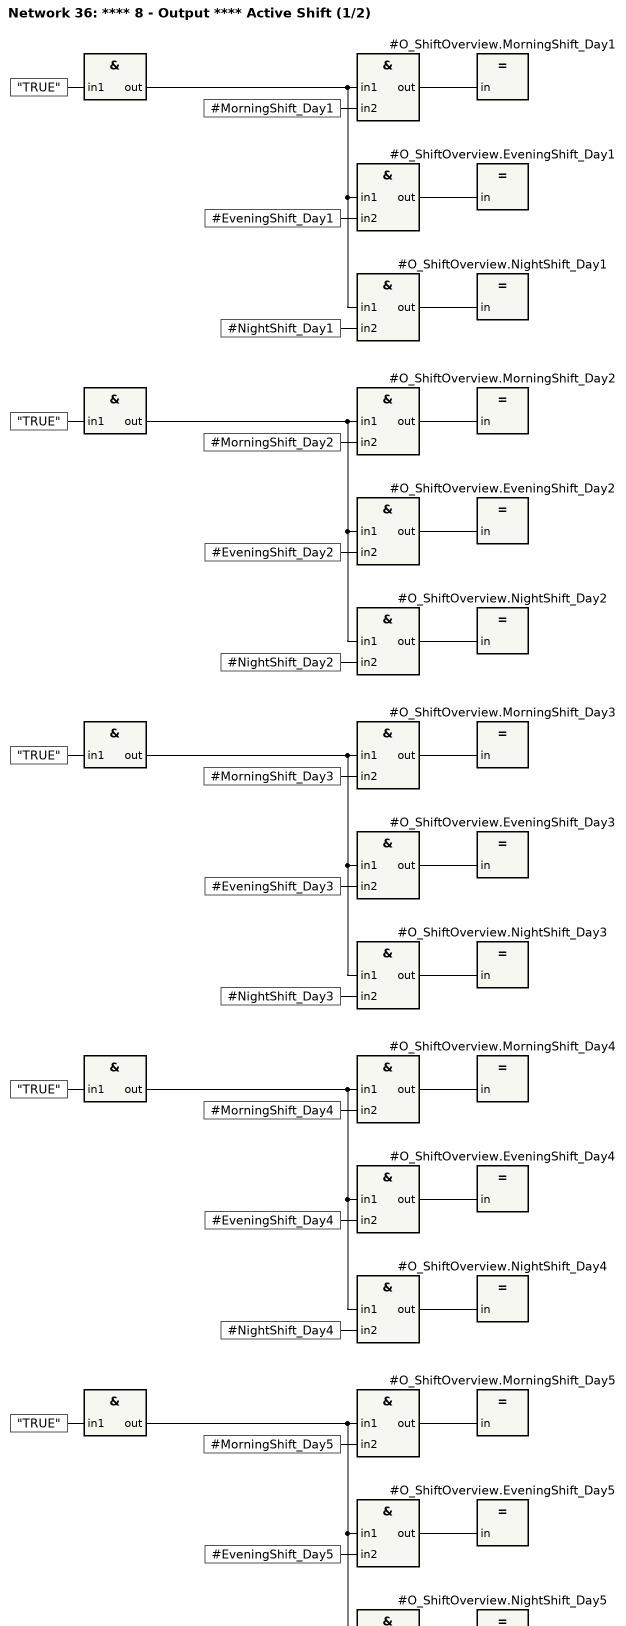
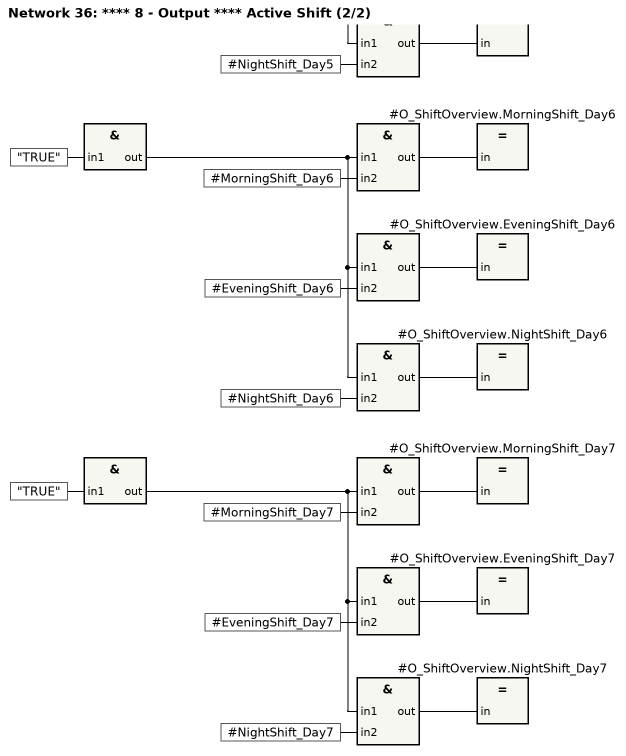
   #O_ShiftOverview.MorningShift_Day1 := "TRUE" AND #MorningShift_Day1;
   #O_ShiftOverview.EveningShift_Day1 := "TRUE" AND #EveningShift_Day1;
   #O_ShiftOverview.NightShift_Day1 := "TRUE" AND #NightShift_Day1;
   #O_ShiftOverview.MorningShift_Day2 := "TRUE" AND #MorningShift_Day2;
   #O_ShiftOverview.EveningShift_Day2 := "TRUE" AND #EveningShift_Day2;
   #O_ShiftOverview.NightShift_Day2 := "TRUE" AND #NightShift_Day2;
   #O_ShiftOverview.MorningShift_Day3 := "TRUE" AND #MorningShift_Day3;
   #O_ShiftOverview.EveningShift_Day3 := "TRUE" AND #EveningShift_Day3;
   #O_ShiftOverview.NightShift_Day3 := "TRUE" AND #NightShift_Day3;
   #O_ShiftOverview.MorningShift_Day4 := "TRUE" AND #MorningShift_Day4;
   #O_ShiftOverview.EveningShift_Day4 := "TRUE" AND #EveningShift_Day4;
   #O_ShiftOverview.NightShift_Day4 := "TRUE" AND #NightShift_Day4;
   #O_ShiftOverview.MorningShift_Day5 := "TRUE" AND #MorningShift_Day5;
   #O_ShiftOverview.EveningShift_Day5 := "TRUE" AND #EveningShift_Day5;
   #O_ShiftOverview.NightShift_Day5 := "TRUE" AND #NightShift_Day5;
   #O_ShiftOverview.MorningShift_Day6 := "TRUE" AND #MorningShift_Day6;
   #O_ShiftOverview.EveningShift_Day6 := "TRUE" AND #EveningShift_Day6;
   #O_ShiftOverview.NightShift_Day6 := "TRUE" AND #NightShift_Day6;
   #O_ShiftOverview.MorningShift_Day7 := "TRUE" AND #MorningShift_Day7;
   #O_ShiftOverview.EveningShift_Day7 := "TRUE" AND #EveningShift_Day7;
   #O_ShiftOverview.NightShift_Day7 := "TRUE" AND #NightShift_Day7;
END_REGION
END_FUNCTION_BLOCK
